(* PLC project v0.6.02_RefactorGateAndTest.project, CODESYS CODESYS V3.5 SP19 Patch 1 *)
(* stored: creationDateTime 2026-08-14T10:10:49.357095, modificationDateTime 2026-08-14T10:10:49.357095 *)

(* values of E_Mode: DISABLE: Mode Désactivé / Veille de sécurité (sorties bloquées); MAINT_N1: Manuel Niveau 1 : Pilotage unitaire avec toutes sécurités actives; MAINT_N2: Manuel Niveau 2 : Pilotage dégradé (droits étendus + bypasses autorisés); SEMI_AUTO: Mode Semi-Automatique (séquenceur automatique) *)

{attribute 'qualified_only'}
{attribute 'strict'}
TYPE E_Mode : (DISABLE := 0, MAINT_N1 := 1, MAINT_N2 := 2, SEMI_AUTO := 3);
END_TYPE

(* values of E_State: DISABLED: Enable faux, neutralisé; INIT: Démarrage / vérifs; READY: Prêt, attend ordre; BUSY: Action en cours; DONE: Action terminée; STOPPING: Décél rampe avant arrêt (StartStop=FALSE ou SafeStop=TRUE) *)

{attribute 'qualified_only'}
{attribute 'strict'}
TYPE E_State : (DISABLED := 0, INIT := 1, READY := 2, BUSY := 3, DONE := 4, STOPPING := 5);
END_TYPE

(* ═══════════════════════════════════════════════════════════════ 🛡️ FB_Encoder_Safety — Bornage physique & relais incohérence redémarrage ─────────────────────────────────────────────────────────────── 📄 Doc métier : DOC/AF/AF_Partie-09_Fonction_Encoder_v2.1.md §3.6/§3.7 DOC/AF/AF_Partie-03_Contrats_Composants_v2.1.md 🎯 Rôle : - Bornage absolu [-99.00 ; +99.00] m (CablePosMSafe gelée sur dernière valeur plausible). - Relais de HomingSuspect (ErrorId bit1). - Expose EncoderIncoherent (= Error) consommé par FB_Modes. ═══════════════════════════════════════════════════════════════ === DECLARATION (à coller dans la partie déclaration du POU FB_Encoder_Safety) === *)
FUNCTION_BLOCK FB_Encoder_Safety
  VAR_INPUT
    Enable : BOOL;  (* Standard *)
    Reset : BOOL;  (* Acquittement défaut (front) — bit0 uniquement (bit1 suit HomingSuspect, voir §7bis) *)
    PowerContactorEngaged : BOOL;  (* Standard *)
    Mode : E_Mode;  (* Standard (contexte, pas encore exploité ce lot) *)
    CablePosM : REAL;  (* Sortie FB_Encoder_Scale DE CE TREUIL *)
    HomingSuspect : BOOL;  (* Sortie FB_Encoder_Homing DE CE TREUIL (§3.7, déjà calculé) *)
    PositionMinM : REAL := -99;  (* Bornage physique dur (Partie10 §3.6) *)
    PositionMaxM : REAL := 99;
    BypassGlobal : BOOL := FALSE;  (* 🌐 Force ErrorId=0, ignore bornage (mise en service) *)
  END_VAR
  VAR_OUTPUT
    Ready : BOOL;
    Busy : BOOL;
    Done : BOOL;
    Error : BOOL;
    ErrorId : WORD;  (* bit0: "Position câble hors plage" - position hors plage physique ; bit1: "Incohérence position boot" - incohérence redémarrage (miroir HomingSuspect) *)
    State : E_State;
    StateAtError : E_State;
    CablePosMSafe : REAL;  (* CablePosM gelée sur dernière valeur plausible si hors plage *)
    EncoderIncoherent : BOOL;  (* = Error — consommé par FB_Modes (refuse SEMI_AUTO) *)
  END_VAR
  VAR
    ResetEdge : R_TRIG;
    ErrorEdge : R_TRIG;
    LastPlausibleCablePosM : REAL;
  END_VAR

            

// === IMPLEMENTATION (à coller dans le corps ST du POU FB_Encoder_Safety) ===

// 🛑 1. GATE — expose la dernière valeur plausible connue même désactivé
IF NOT Enable THEN
    Ready := FALSE; Busy := FALSE; Done := FALSE;
    State := E_State.DISABLED;
    CablePosMSafe := LastPlausibleCablePosM;
    EncoderIncoherent := FALSE;
    RETURN;
END_IF;

Ready := TRUE;
State := E_State.READY;

// 🔑 2. RESET FRONT
ResetEdge(CLK := Reset);

// 🌐 BYPASS GLOBAL : force ErrorId = 0, ignore bornage et incohérence
IF BypassGlobal THEN
    ErrorId := 16#0000;
END_IF;

// 🔍 3. BORNAGE PHYSIQUE ABSOLU (§3.6) — bit0
IF NOT BypassGlobal AND ((CablePosM < PositionMinM) OR (CablePosM > PositionMaxM)) THEN
    ErrorId := ErrorId OR 16#0001;
ELSE
    ErrorId := ErrorId AND 16#FFFE; (* Auto-clearing dès que la position revient dans la plage valide *)
END_IF;

// 🔍 4. RELAIS INCOHÉRENCE REDÉMARRAGE (§3.7, calculée par FB_Encoder_Homing) — bit1
// Pas d'acquittement ici : la levée se fait via BtnConfirmCoherence/nouveau Home côté
// FB_Encoder_Homing (source), ce FB ne fait QUE relayer l'information pour FB_Modes.
IF NOT BypassGlobal THEN
    IF HomingSuspect THEN
        ErrorId := ErrorId OR 16#0002;
    ELSE
        ErrorId := ErrorId AND 16#FFFD;
    END_IF;
END_IF;

// 🧊 5. GELER SUR DOUTE (§6) — CablePosMSafe ne suit PAS CablePosM si hors plage
IF (ErrorId AND 16#0001) = 16#0000 THEN
    LastPlausibleCablePosM := CablePosM;
END_IF;
CablePosMSafe := LastPlausibleCablePosM;

// 📤 6. SORTIES ÉTAT
Error := (ErrorId <> 16#0000);
ErrorEdge(CLK := Error);
IF ErrorEdge.Q THEN
    StateAtError := State;
END_IF;

EncoderIncoherent := Error;
Busy := FALSE;
Done := FALSE;

          
END_FUNCTION_BLOCK
